FUNCTION TryConvert_REAL_TO_BYTE : BOOL
VAR_INPUT
	in : REAL;
	out : REFERENCE TO BYTE;
END_VAR

IF in > DatatypeLimits.MAX_VALUE_OF_REAL_WHICH_CAN_BE_HELD_IN_A_BYTE THEN
	RETURN;
END_IF

IF in < DatatypeLimits.MIN_VALUE_OF_REAL_WHICH_CAN_BE_HELD_IN_A_BYTE THEN
	RETURN;
END_IF

out := REAL_TO_BYTE(in);
TryConvert_REAL_TO_BYTE := TRUE;

END_FUNCTION

(* stored: Version 1.1.0.1, ProductVersion 3.1.4024.12
   POU TryConvert_REAL_TO_BYTE: Id {18379508-55d2-4515-b193-68c93962e584}, SpecialFunc None *)
